TYPE ST_CoeEntry_SINT EXTENDS ST_CoeEntry :
STRUCT
	Value	: SINT;
END_STRUCT
END_TYPE

(* stored: Version 1.1.0.1, ProductVersion 3.1.4024.14
   DUT ST_CoeEntry_SINT: Id {703e0e14-89de-03f6-02e4-c2189681bf7a} *)
